{attribute 'linkalways'} 
{attribute 'no_explicit_call' := 'This FB is a CLASS and must be accessed using methods or properties'}
{attribute 'enable_dynamic_creation'}
FUNCTION_BLOCK Node_F_VN_SetAt_TcVnPoint3_LREAL EXTENDS VisionNode
VAR
    aElement : _TcVnPoint3_LREAL;
    ipContainer : _ITcVnContainer;
    nIndex : _ULINT(0);
    hrPrev : _HRESULT(S_OK);
    hresult : _HRESULT(S_OK);
END_VAR

METHOD PUBLIC  Clone : I_Node
VAR
	pNode : POINTER TO Node_F_VN_SetAt_TcVnPoint3_LREAL;
END_VAR
pNode := __NEW(Node_F_VN_SetAt_TcVnPoint3_LREAL);
Clone := pNode^;
END_METHOD

METHOD FB_init : BOOL
VAR_INPUT
	bInitRetains : BOOL; // if TRUE, the retain variables are initialized (warm start / cold start)
	bInCopyCode : BOOL;  // if TRUE, the instance afterwards gets moved into the copy code (online change)
END_VAR
AddInput('aElement', aElement);
AddInput('ipContainer', ipContainer);
AddInput('nIndex', nIndex);
AddInput('hrPrev', hrPrev);
AddOutput('ipContainer', ipContainer);
AddOutput('hresult',hresult);
END_METHOD

METHOD PROTECTED OnExecute : HRESULT
hresult.Value := F_VN_SetAt_TcVnPoint3_LREAL(
    aElement := aElement.Value,
    ipContainer := ipContainer.Value,
    nIndex := nIndex.Value,
    hrPrev:= hrPrev.Value);
END_METHOD

METHOD PUBLIC PreExecutionCheck
VAR_INPUT
	Check : I_PreExecutionChecks;
END_VAR
Check.IsTrue(ipContainer.IsValid, 'ipContainer must be a valid container');
END_METHOD

END_FUNCTION_BLOCK

(* stored: Version 1.1.0.1, ProductVersion 3.1.4024.13
   POU Node_F_VN_SetAt_TcVnPoint3_LREAL: Id {c44efc57-63ff-4273-b147-b728cda96e81}, SpecialFunc None
   Folder Constructor: Id {2d0a2e2f-e298-4f2f-af50-62a5c580faa8}
   Method Clone: Id {e95be4de-cffc-42ab-abbc-81b2483b0ee2}
   Method FB_init: Id {1414546b-a980-4cfa-b39c-43e18eae0564}
   Method OnExecute: Id {51d58fe5-e288-4098-92eb-ed57cb142533}
   Method PreExecutionCheck: Id {450ed004-9c73-4507-8ef2-0197309e594a} *)
